Staubli VAL3: getAction.pgx

public program getAction(string& x_sInstruction[], bool x_bType, num x_nIndex)
  local string l_sInstruction
begin
  // get the instruction and fill as an array
  if x_nIndex>=0
    if x_bType
      // take gun ON
      l_sInstruction=saveTool:sActionON[x_nIndex]
    else
      // take gun OFF
      l_sInstruction=saveTool:sActionOFF[x_nIndex]
    endIf
    // make it to three element
    if l_sInstruction==""
      l_sInstruction=",,"
    endIf
    call use:stringToArray(l_sInstruction,x_sInstruction)
  endIf
end
